Staubli VAL3: TestSetmoveid.pgx

program TestSetmoveid()
  local num l_nIndex
begin
  //清空运动堆栈中已有运动指令，会自动把moveid设置为0
  resetMotion()


  //清除屏幕
  cls()

  //强制设置到用户界面
  userPage()

  //设置moveid
  setMoveId(-1000.15)

  //循环语句
  for l_nIndex=0 to 100
    mMdesc.blend=off
    movej(jJ,tTool,mMdesc)


    gotoxy(0,0)
    put("MOVEID的值是:"+toString(".3",getMoveId()))
  endFor
  waitEndMove()




end
